TYPE (* Typedef of the TP CAN Message *)
  (* Version 1.0, 2025-09-04, franz *)
  PACKAGE isobus;
  CAN_MSG_TP : STRUCT
    data : ARRAY [*] OF BYTE;
  END_STRUCT;
END_TYPE
